// SIMATIC S7-200 SMART project (STEP 7-Micro/WIN SMART), CPU ST60

SYMBOL_TABLE V区符号
参数传输成功           V0.0     // 接收工控机传来的数据传输成功信号
参数是否更新           V0.1
挡板自动控制完成标志       V0.2
挡板电机开关           V0.3
挡板手动向内           V0.4
挡板手动向外           V0.5
置工件就绪            V0.6
下料电机开关           V0.7
下料前进点动           V1.0
下料后退点动           V1.1
冷却电机开关           V1.2
冷却电机向内           V1.3
冷却电机向外           V1.4
挡板电机查找原点按钮       V11.1
下料电机查找原点按钮       V11.2
冷却电机查找原点按钮       V11.3
挡板自动控制           V11.4
下料下移一个工位         V11.5
下料启动按钮           V11.6
下料手动完成标志         V11.7
回到底部             V12.0
冷却自动控制           V12.1
挡板电机初始化完成位       V20.1
挡板电机当前运动方向       V20.2
挡板电机查找原点完成位      V20.3
挡板电机GOTO完成位      V20.4
挡板电机错误参数         VB21
挡板电机当前位置         VD24
挡板电机当前速度         VD28
挡板电机移动位置         VD44
挡板电机速度           VD48
挡板电机移动模式         VB41
挡板电机停止运动轴        V40.1
挡板电机运动方向         V40.2
冷却电机初始化完成位       V60.1
冷却电机当前运动方向       V60.2
冷却电机查找原点完成位      V60.3
冷却电机GOTO完成位      V60.4
冷却电机错误参数         VB61
冷却电机当前位置         VD64
冷却电机当前速度         VD68
冷却电机移动位置         VD84
冷却电机速度           VD88
冷却电机移动模式         VB81
冷却电机停止运动轴        V80.1
冷却电机运动方向         V80.2
下料电机初始化完成位       V100.1
下料电机当前运动方向       V100.2
下料电机查找原点完成位      V100.3
下料电机GOTO完成位      V100.4
下料电机错误参数         VB101
下料电机当前位置         VD104
下料电机当前速度         VD108
下料电机移动位置         VD124
下料电机速度           VD128
下料电机移动模式         VB121
下料电机停止运动轴        V120.1
下料电机运动方向         V120.2
下料电机运动到杆件放置      VD150
下料电机下移一个杆件位      VD154
下料电机一号杆件位置       VD158
下料电机二号杆件位置       VD162
下料电机三号杆件位置       VD166
下料电机四号杆件位置       VD170
下料电机五号杆件位置       VD174
下料电机运动到下料位置      VD178
上一杆件数据           VD140
当前杆件数据           VD144
END_SYMBOL_TABLE

SYMBOL_TABLE 系统符号
Always_On        SM0.0    // 始终接通
END_SYMBOL_TABLE

SYMBOL_TABLE M区符号
挡板超限报警           M0.0     // 挡板的位置超过左右极限传感器的位置
更新配对表            M0.1
电机是否就绪状态位        M0.3
上料步进到位状态位        M0.4
上料工件有无状态位        M0.5
下料步进到位状态位        M0.6
下料小车到位状态位        M0.7
步进报警信息           M1.0
上料传动故障报警         M1.1
两次杆件之差           MD12
END_SYMBOL_TABLE

ORGANIZATION_BLOCK 主程序:OB1
TITLE=
BEGIN
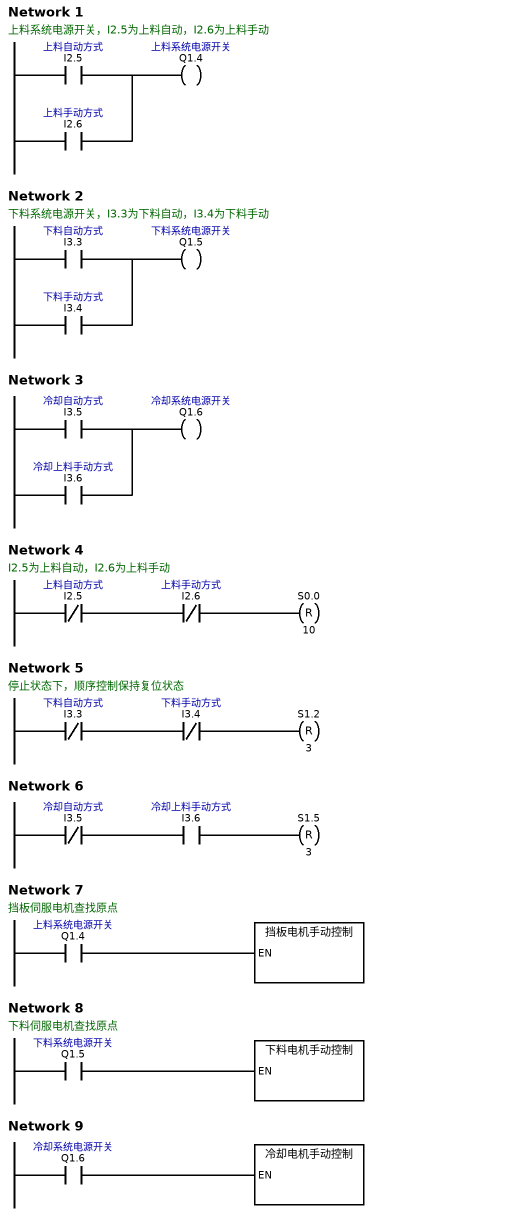
Network 1
// 上料系统电源开关，I2.5为上料自动，I2.6为上料手动
LD     上料自动方式:I2.5
O      上料手动方式:I2.6
=      上料系统电源开关:Q1.4
Network 2
// 下料系统电源开关，I3.3为下料自动，I3.4为下料手动
LD     下料自动方式:I3.3
O      下料手动方式:I3.4
=      下料系统电源开关:Q1.5
Network 3
LD     冷却自动方式:I3.5
O      冷却上料手动方式:I3.6
=      冷却系统电源开关:Q1.6
Network 4
// I2.5为上料自动，I2.6为上料手动
LDN    上料自动方式:I2.5
AN     上料手动方式:I2.6
R      S0.0, 10
Network 5
// 停止状态下，顺序控制保持复位状态
LDN    下料自动方式:I3.3
AN     下料手动方式:I3.4
R      S1.2, 3
Network 6
LDN    冷却自动方式:I3.5
A      冷却上料手动方式:I3.6
R      S1.5, 3
Network 7
// 挡板伺服电机查找原点
LD     上料系统电源开关:Q1.4
CALL   挡板电机手动控制:SBR7
Network 8
// 下料伺服电机查找原点
LD     下料系统电源开关:Q1.5
CALL   下料电机手动控制:SBR9
Network 9
LD     冷却系统电源开关:Q1.6
CALL   冷却电机手动控制:SBR18
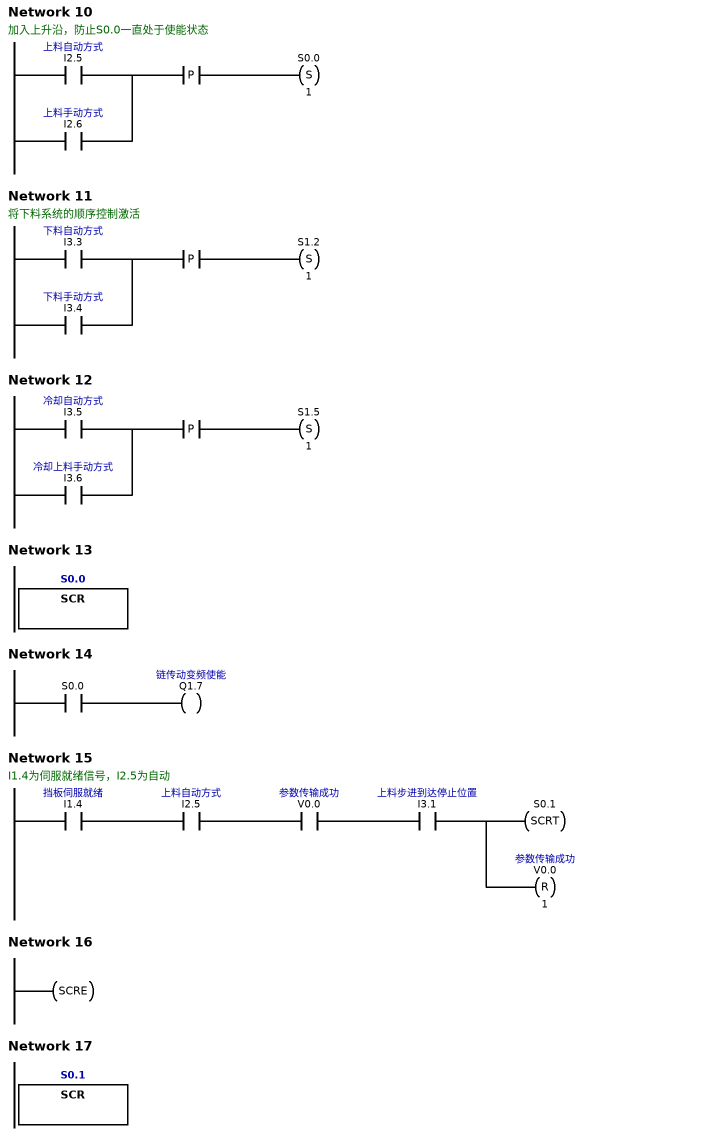
Network 10
// 加入上升沿，防止S0.0一直处于使能状态
LD     上料自动方式:I2.5
O      上料手动方式:I2.6
EU
S      S0.0, 1
Network 11
// 将下料系统的顺序控制激活
LD     下料自动方式:I3.3
O      下料手动方式:I3.4
EU
S      S1.2, 1
Network 12
LD     冷却自动方式:I3.5
O      冷却上料手动方式:I3.6
EU
S      S1.5, 1
Network 13
LSCR   S0.0
Network 14
LD     S0.0
=      链传动变频使能:Q1.7
Network 15
// I1.4为伺服就绪信号，I2.5为自动
LD     挡板伺服就绪:I1.4
A      上料自动方式:I2.5
A      参数传输成功:V0.0
A      上料步进到达停止位置:I3.1
SCRT   S0.1
R      参数传输成功:V0.0, 1
Network 16
SCRE
Network 17
LSCR   S0.1
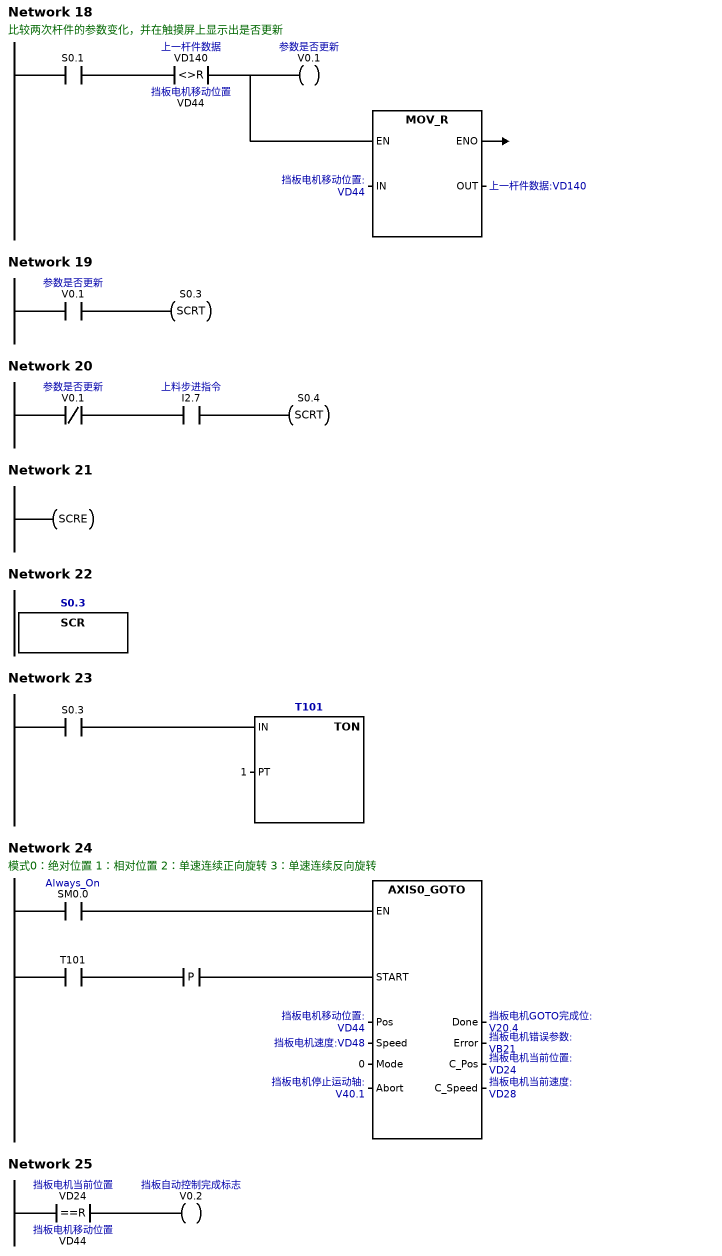
Network 18
// 比较两次杆件的参数变化，并在触摸屏上显示出是否更新
LD     S0.1
AR<>   上一杆件数据:VD140, 挡板电机移动位置:VD44
=      参数是否更新:V0.1
MOVR   挡板电机移动位置:VD44, 上一杆件数据:VD140
Network 19
LD     参数是否更新:V0.1
SCRT   S0.3
Network 20
LDN    参数是否更新:V0.1
A      上料步进指令:I2.7
SCRT   S0.4
Network 21
SCRE
Network 22
LSCR   S0.3
Network 23
LD     S0.3
TON    T101, 1
Network 24
// 模式0：绝对位置 1：相对位置 2：单速连续正向旋转 3：单速连续反向旋转
LD     Always_On:SM0.0
=      L60.0
LD     T101
EU
=      L63.7
LD     L60.0
CALL   AXIS0_GOTO:SBR4, L63.7, 挡板电机移动位置:VD44, 挡板电机速度:VD48, 0, 挡板电机停止运动轴:V40.1, 挡板电机GOTO完成位:V20.4, 挡板电机错误参数:VB21, 挡板电机当前位置:VD24, 挡板电机当前速度:VD28
Network 25
LDR=   挡板电机当前位置:VD24, 挡板电机移动位置:VD44
=      挡板自动控制完成标志:V0.2
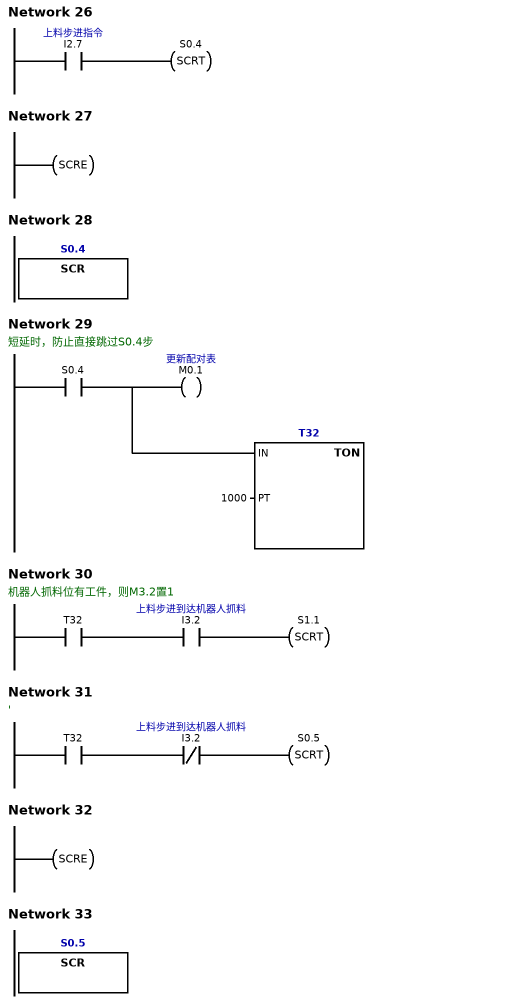
Network 26
LD     上料步进指令:I2.7
SCRT   S0.4
Network 27
SCRE
Network 28
LSCR   S0.4
Network 29
// 短延时，防止直接跳过S0.4步
LD     S0.4
=      更新配对表:M0.1
TON    T32, 1000
Network 30
// 机器人抓料位有工件，则M3.2置1
LD     T32
A      上料步进到达机器人抓料:I3.2
SCRT   S1.1
Network 31
// '
LD     T32
AN     上料步进到达机器人抓料:I3.2
SCRT   S0.5
Network 32
SCRE
Network 33
LSCR   S0.5
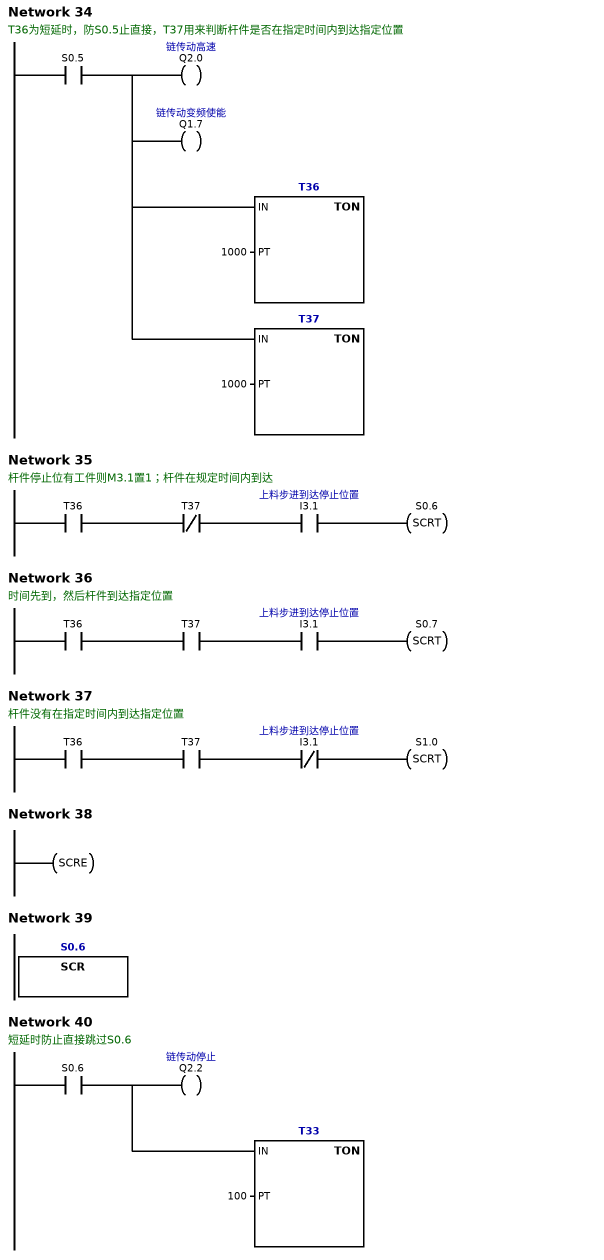
Network 34
// T36为短延时，防S0.5止直接，T37用来判断杆件是否在指定时间内到达指定位置
LD     S0.5
=      链传动高速:Q2.0
=      链传动变频使能:Q1.7
TON    T36, 1000
TON    T37, 1000
Network 35
// 杆件停止位有工件则M3.1置1；杆件在规定时间内到达
LD     T36
AN     T37
A      上料步进到达停止位置:I3.1
SCRT   S0.6
Network 36
// 时间先到，然后杆件到达指定位置
LD     T36
A      T37
A      上料步进到达停止位置:I3.1
SCRT   S0.7
Network 37
// 杆件没有在指定时间内到达指定位置
LD     T36
A      T37
AN     上料步进到达停止位置:I3.1
SCRT   S1.0
Network 38
SCRE
Network 39
LSCR   S0.6
Network 40
// 短延时防止直接跳过S0.6
LD     S0.6
=      链传动停止:Q2.2
TON    T33, 100
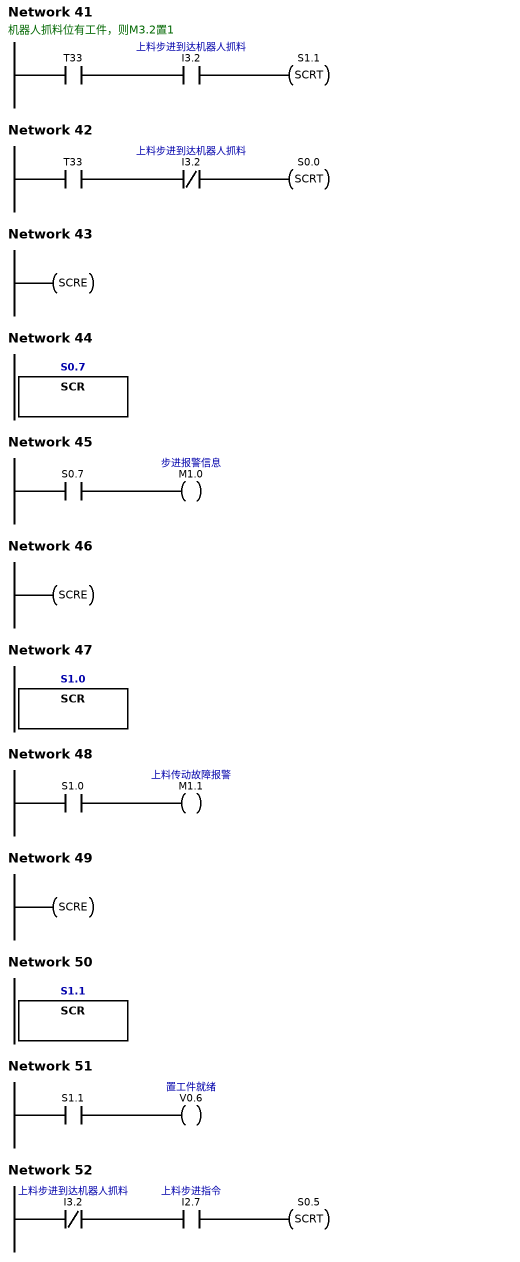
Network 41
// 机器人抓料位有工件，则M3.2置1
LD     T33
A      上料步进到达机器人抓料:I3.2
SCRT   S1.1
Network 42
LD     T33
AN     上料步进到达机器人抓料:I3.2
SCRT   S0.0
Network 43
SCRE
Network 44
LSCR   S0.7
Network 45
LD     S0.7
=      步进报警信息:M1.0
Network 46
SCRE
Network 47
LSCR   S1.0
Network 48
LD     S1.0
=      上料传动故障报警:M1.1
Network 49
SCRE
Network 50
LSCR   S1.1
Network 51
LD     S1.1
=      置工件就绪:V0.6
Network 52
LDN    上料步进到达机器人抓料:I3.2
A      上料步进指令:I2.7
SCRT   S0.5
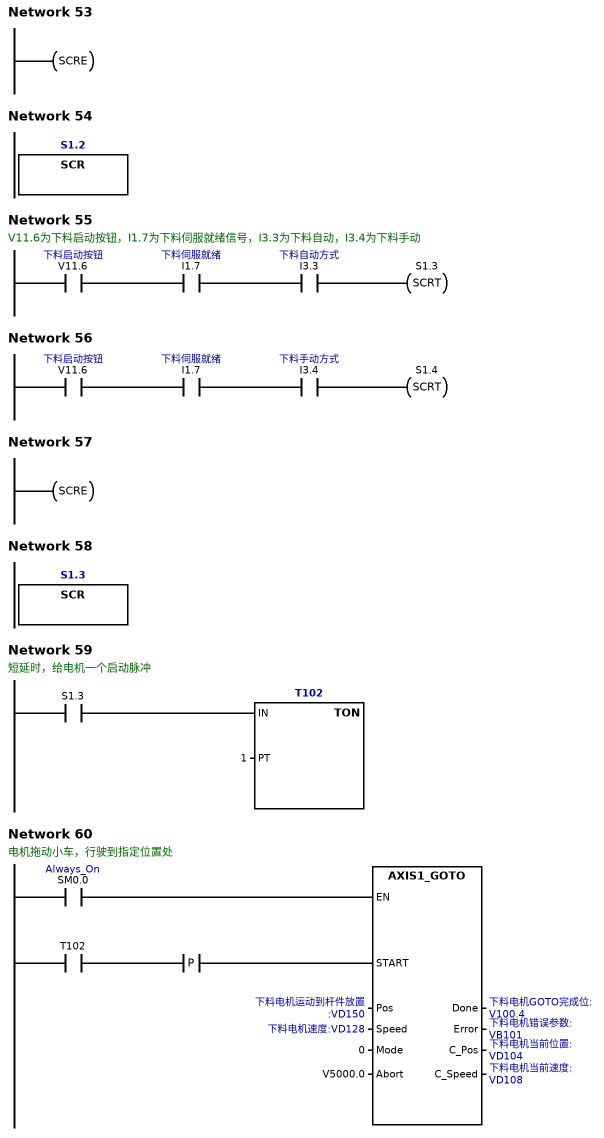
Network 53
SCRE
Network 54
LSCR   S1.2
Network 55
// V11.6为下料启动按钮，I1.7为下料伺服就绪信号，I3.3为下料自动，I3.4为下料手动
LD     下料启动按钮:V11.6
A      下料伺服就绪:I1.7
A      下料自动方式:I3.3
SCRT   S1.3
Network 56
LD     下料启动按钮:V11.6
A      下料伺服就绪:I1.7
A      下料手动方式:I3.4
SCRT   S1.4
Network 57
SCRE
Network 58
LSCR   S1.3
Network 59
// 短延时，给电机一个启动脉冲
LD     S1.3
TON    T102, 1
Network 60
// 电机拖动小车，行驶到指定位置处
LD     Always_On:SM0.0
=      L60.0
LD     T102
EU
=      L63.7
LD     L60.0
CALL   AXIS1_GOTO:SBR11, L63.7, 下料电机运动到杆件放置:VD150, 下料电机速度:VD128, 0, V5000.0, 下料电机GOTO完成位:V100.4, 下料电机错误参数:VB101, 下料电机当前位置:VD104, 下料电机当前速度:VD108
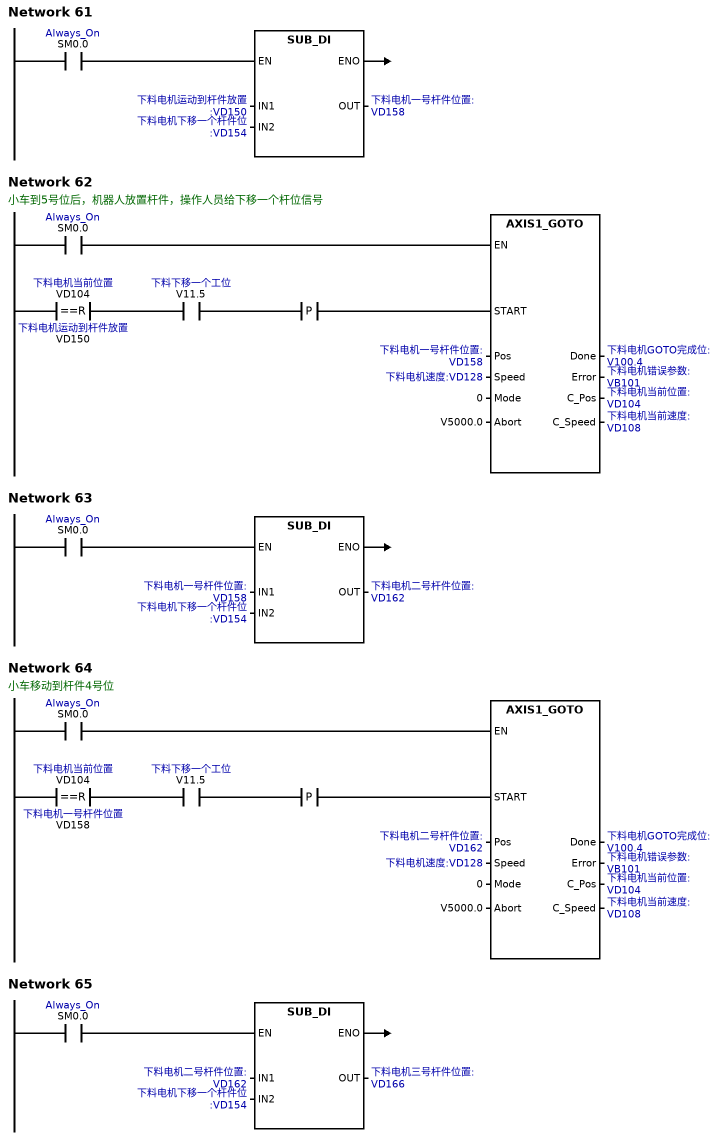
Network 61
LD     Always_On:SM0.0
MOVD   下料电机运动到杆件放置:VD150, 下料电机一号杆件位置:VD158
-D     下料电机下移一个杆件位:VD154, 下料电机一号杆件位置:VD158
Network 62
// 小车到5号位后，机器人放置杆件，操作人员给下移一个杆位信号
LD     Always_On:SM0.0
=      L60.0
LDR=   下料电机当前位置:VD104, 下料电机运动到杆件放置:VD150
A      下料下移一个工位:V11.5
EU
=      L63.7
LD     L60.0
CALL   AXIS1_GOTO:SBR11, L63.7, 下料电机一号杆件位置:VD158, 下料电机速度:VD128, 0, V5000.0, 下料电机GOTO完成位:V100.4, 下料电机错误参数:VB101, 下料电机当前位置:VD104, 下料电机当前速度:VD108
Network 63
LD     Always_On:SM0.0
MOVD   下料电机一号杆件位置:VD158, 下料电机二号杆件位置:VD162
-D     下料电机下移一个杆件位:VD154, 下料电机二号杆件位置:VD162
Network 64
// 小车移动到杆件4号位
LD     Always_On:SM0.0
=      L60.0
LDR=   下料电机当前位置:VD104, 下料电机一号杆件位置:VD158
A      下料下移一个工位:V11.5
EU
=      L63.7
LD     L60.0
CALL   AXIS1_GOTO:SBR11, L63.7, 下料电机二号杆件位置:VD162, 下料电机速度:VD128, 0, V5000.0, 下料电机GOTO完成位:V100.4, 下料电机错误参数:VB101, 下料电机当前位置:VD104, 下料电机当前速度:VD108
Network 65
LD     Always_On:SM0.0
MOVD   下料电机二号杆件位置:VD162, 下料电机三号杆件位置:VD166
-D     下料电机下移一个杆件位:VD154, 下料电机三号杆件位置:VD166
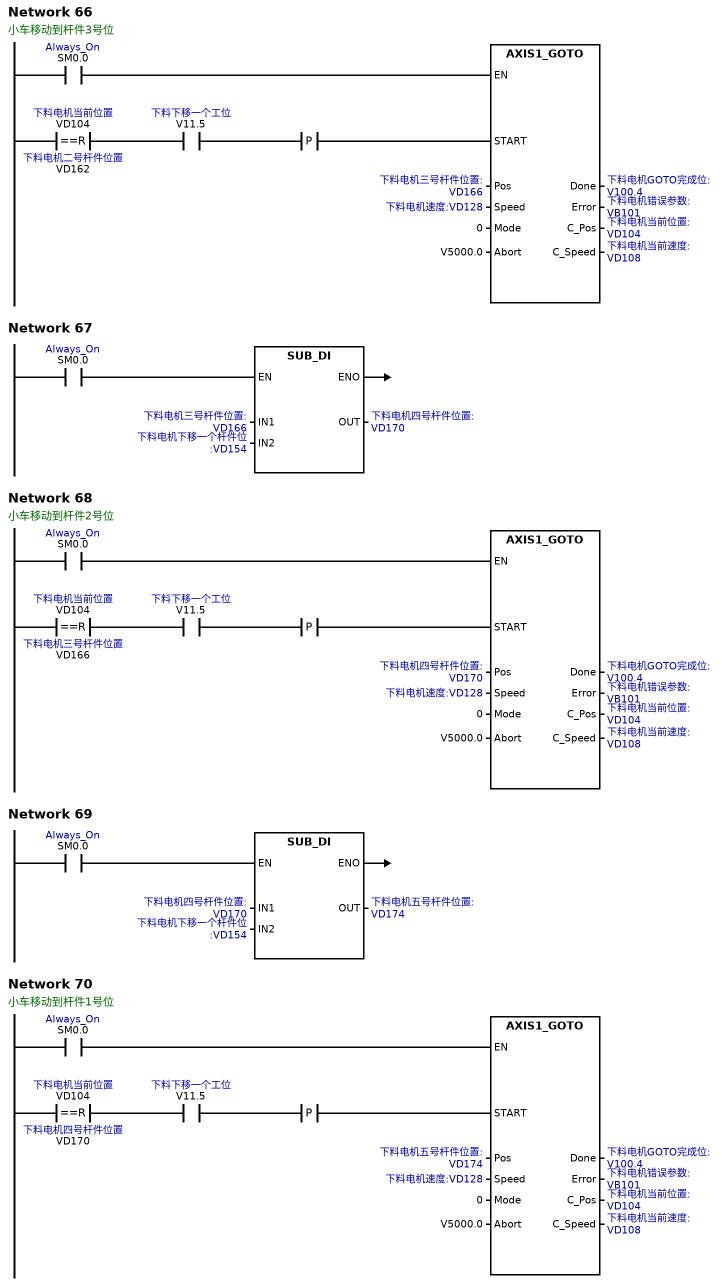
Network 66
// 小车移动到杆件3号位
LD     Always_On:SM0.0
=      L60.0
LDR=   下料电机当前位置:VD104, 下料电机二号杆件位置:VD162
A      下料下移一个工位:V11.5
EU
=      L63.7
LD     L60.0
CALL   AXIS1_GOTO:SBR11, L63.7, 下料电机三号杆件位置:VD166, 下料电机速度:VD128, 0, V5000.0, 下料电机GOTO完成位:V100.4, 下料电机错误参数:VB101, 下料电机当前位置:VD104, 下料电机当前速度:VD108
Network 67
LD     Always_On:SM0.0
MOVD   下料电机三号杆件位置:VD166, 下料电机四号杆件位置:VD170
-D     下料电机下移一个杆件位:VD154, 下料电机四号杆件位置:VD170
Network 68
// 小车移动到杆件2号位
LD     Always_On:SM0.0
=      L60.0
LDR=   下料电机当前位置:VD104, 下料电机三号杆件位置:VD166
A      下料下移一个工位:V11.5
EU
=      L63.7
LD     L60.0
CALL   AXIS1_GOTO:SBR11, L63.7, 下料电机四号杆件位置:VD170, 下料电机速度:VD128, 0, V5000.0, 下料电机GOTO完成位:V100.4, 下料电机错误参数:VB101, 下料电机当前位置:VD104, 下料电机当前速度:VD108
Network 69
LD     Always_On:SM0.0
MOVD   下料电机四号杆件位置:VD170, 下料电机五号杆件位置:VD174
-D     下料电机下移一个杆件位:VD154, 下料电机五号杆件位置:VD174
Network 70
// 小车移动到杆件1号位
LD     Always_On:SM0.0
=      L60.0
LDR=   下料电机当前位置:VD104, 下料电机四号杆件位置:VD170
A      下料下移一个工位:V11.5
EU
=      L63.7
LD     L60.0
CALL   AXIS1_GOTO:SBR11, L63.7, 下料电机五号杆件位置:VD174, 下料电机速度:VD128, 0, V5000.0, 下料电机GOTO完成位:V100.4, 下料电机错误参数:VB101, 下料电机当前位置:VD104, 下料电机当前速度:VD108
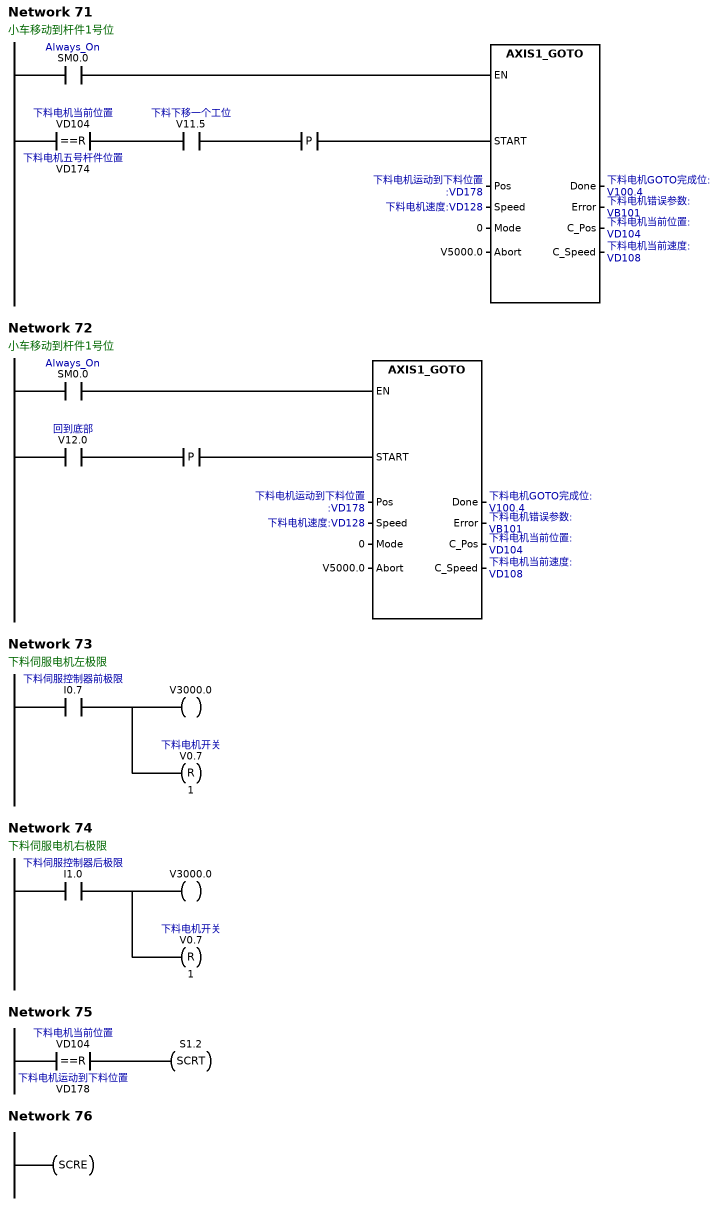
Network 71
// 小车移动到杆件1号位
LD     Always_On:SM0.0
=      L60.0
LDR=   下料电机当前位置:VD104, 下料电机五号杆件位置:VD174
A      下料下移一个工位:V11.5
EU
=      L63.7
LD     L60.0
CALL   AXIS1_GOTO:SBR11, L63.7, 下料电机运动到下料位置:VD178, 下料电机速度:VD128, 0, V5000.0, 下料电机GOTO完成位:V100.4, 下料电机错误参数:VB101, 下料电机当前位置:VD104, 下料电机当前速度:VD108
Network 72
// 小车移动到杆件1号位
LD     Always_On:SM0.0
=      L60.0
LD     回到底部:V12.0
EU
=      L63.7
LD     L60.0
CALL   AXIS1_GOTO:SBR11, L63.7, 下料电机运动到下料位置:VD178, 下料电机速度:VD128, 0, V5000.0, 下料电机GOTO完成位:V100.4, 下料电机错误参数:VB101, 下料电机当前位置:VD104, 下料电机当前速度:VD108
Network 73
// 下料伺服电机左极限
LD     下料伺服控制器前极限:I0.7
=      V3000.0
R      下料电机开关:V0.7, 1
Network 74
// 下料伺服电机右极限
LD     下料伺服控制器后极限:I1.0
=      V3000.0
R      下料电机开关:V0.7, 1
Network 75
LDR=   下料电机当前位置:VD104, 下料电机运动到下料位置:VD178
SCRT   S1.2
Network 76
SCRE
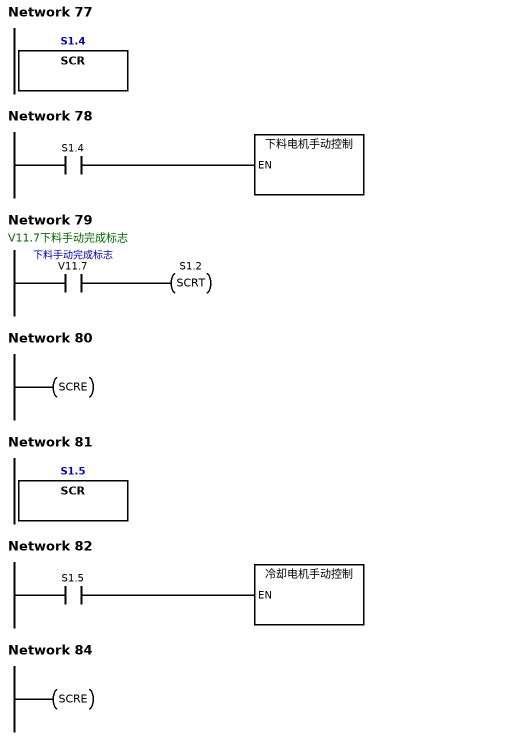
Network 77
LSCR   S1.4
Network 78
LD     S1.4
CALL   下料电机手动控制:SBR9
Network 79
// V11.7下料手动完成标志
LD     下料手动完成标志:V11.7
SCRT   S1.2
Network 80
SCRE
Network 81
LSCR   S1.5
Network 82
LD     S1.5
CALL   冷却电机手动控制:SBR18
Network 84
SCRE
END_ORGANIZATION_BLOCK

// SBR2: protected block, not included

// SBR3: protected block, not included

// SBR4: protected block, not included

// SBR5: protected block, not included

// SBR6: protected block, not included

SUBROUTINE_BLOCK 挡板电机手动控制:SBR7
TITLE=子程序注释
BEGIN
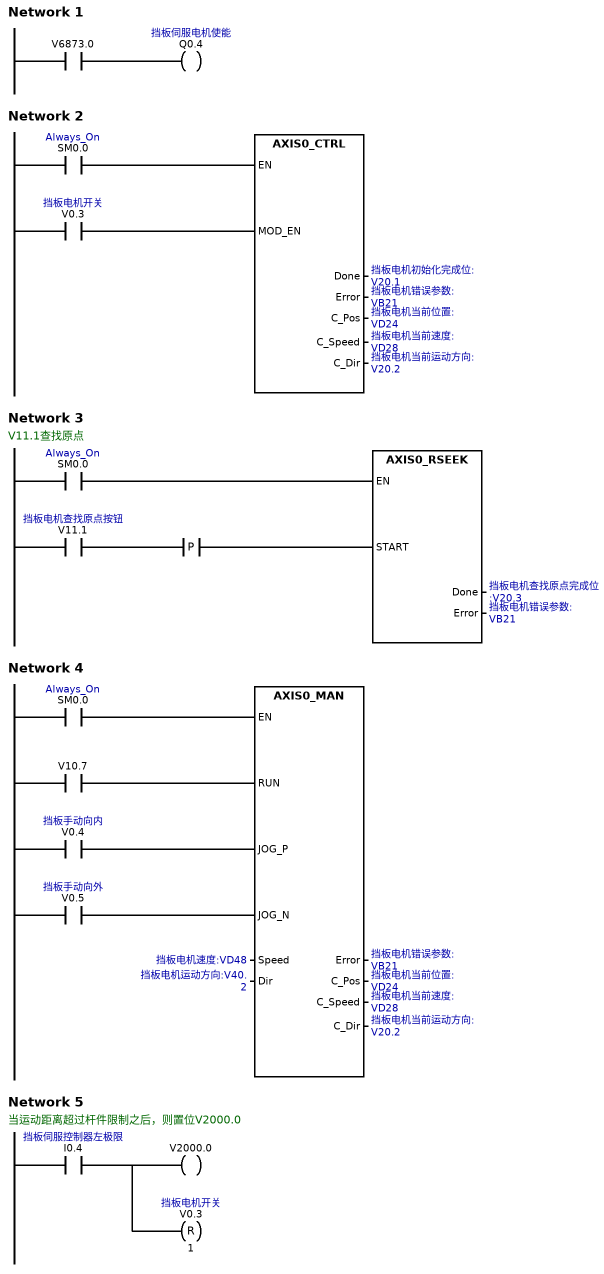
Network 1
LD     V6873.0
=      挡板伺服电机使能:Q0.4
Network 2
LD     Always_On:SM0.0
=      L60.0
LD     挡板电机开关:V0.3
=      L63.7
LD     L60.0
CALL   AXIS0_CTRL:SBR2, L63.7, 挡板电机初始化完成位:V20.1, 挡板电机错误参数:VB21, 挡板电机当前位置:VD24, 挡板电机当前速度:VD28, 挡板电机当前运动方向:V20.2
Network 3
// V11.1查找原点
LD     Always_On:SM0.0
=      L60.0
LD     挡板电机查找原点按钮:V11.1
EU
=      L63.7
LD     L60.0
CALL   AXIS0_RSEEK:SBR5, L63.7, 挡板电机查找原点完成位:V20.3, 挡板电机错误参数:VB21
Network 4
LD     Always_On:SM0.0
=      L60.0
LD     V10.7
=      L63.7
LD     挡板手动向内:V0.4
=      L63.6
LD     挡板手动向外:V0.5
=      L63.5
LD     L60.0
CALL   AXIS0_MAN:SBR3, L63.7, L63.6, L63.5, 挡板电机速度:VD48, 挡板电机运动方向:V40.2, 挡板电机错误参数:VB21, 挡板电机当前位置:VD24, 挡板电机当前速度:VD28, 挡板电机当前运动方向:V20.2
Network 5
// 当运动距离超过杆件限制之后，则置位V2000.0
LD     挡板伺服控制器左极限:I0.4
=      V2000.0
R      挡板电机开关:V0.3, 1
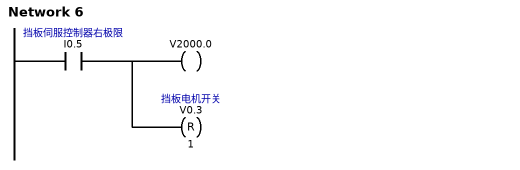
Network 6
LD     挡板伺服控制器右极限:I0.5
=      V2000.0
R      挡板电机开关:V0.3, 1
END_SUBROUTINE_BLOCK

SUBROUTINE_BLOCK 下料电机手动控制:SBR9
TITLE=子程序注释
BEGIN
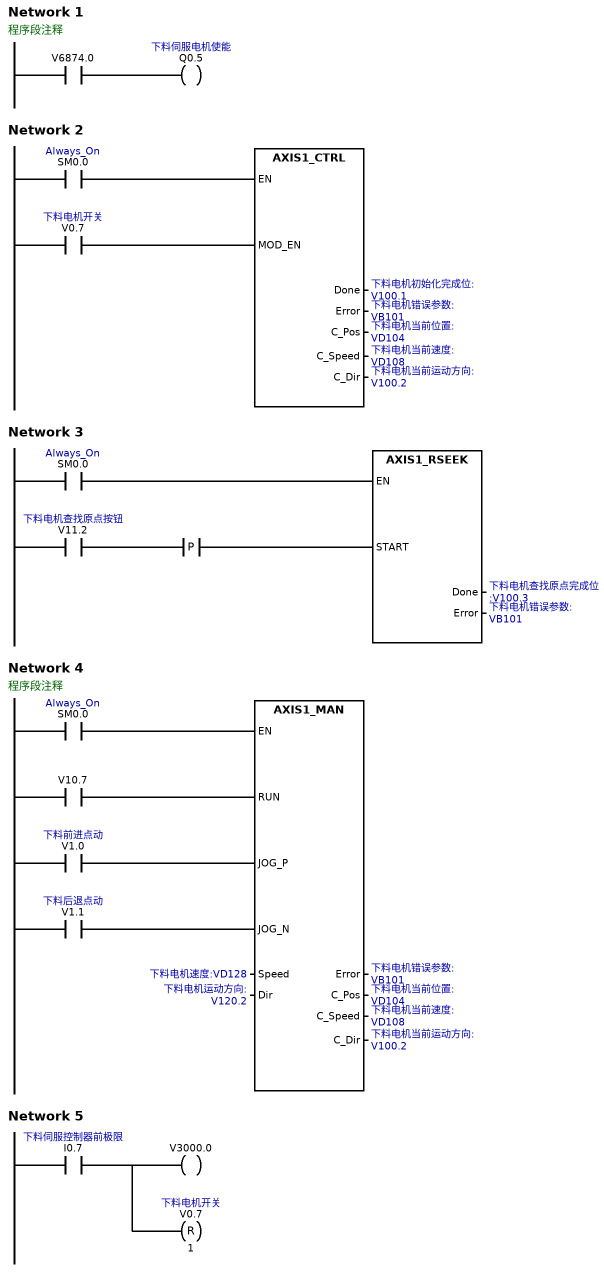
Network 1
// 程序段注释
LD     V6874.0
=      下料伺服电机使能:Q0.5
Network 2
LD     Always_On:SM0.0
=      L60.0
LD     下料电机开关:V0.7
=      L63.7
LD     L60.0
CALL   AXIS1_CTRL:SBR6, L63.7, 下料电机初始化完成位:V100.1, 下料电机错误参数:VB101, 下料电机当前位置:VD104, 下料电机当前速度:VD108, 下料电机当前运动方向:V100.2
Network 3
LD     Always_On:SM0.0
=      L60.0
LD     下料电机查找原点按钮:V11.2
EU
=      L63.7
LD     L60.0
CALL   AXIS1_RSEEK:SBR12, L63.7, 下料电机查找原点完成位:V100.3, 下料电机错误参数:VB101
Network 4
// 程序段注释
LD     Always_On:SM0.0
=      L60.0
LD     V10.7
=      L63.7
LD     下料前进点动:V1.0
=      L63.6
LD     下料后退点动:V1.1
=      L63.5
LD     L60.0
CALL   AXIS1_MAN:SBR10, L63.7, L63.6, L63.5, 下料电机速度:VD128, 下料电机运动方向:V120.2, 下料电机错误参数:VB101, 下料电机当前位置:VD104, 下料电机当前速度:VD108, 下料电机当前运动方向:V100.2
Network 5
LD     下料伺服控制器前极限:I0.7
=      V3000.0
R      下料电机开关:V0.7, 1
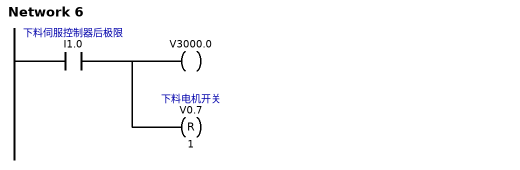
Network 6
LD     下料伺服控制器后极限:I1.0
=      V3000.0
R      下料电机开关:V0.7, 1
END_SUBROUTINE_BLOCK

// SBR10: protected block, not included

// SBR11: protected block, not included

// SBR12: protected block, not included

// SBR13: protected block, not included

// SBR14: protected block, not included

// SBR15: protected block, not included

// SBR16: protected block, not included

SUBROUTINE_BLOCK 冷却电机手动控制:SBR18
TITLE=子程序注释
BEGIN
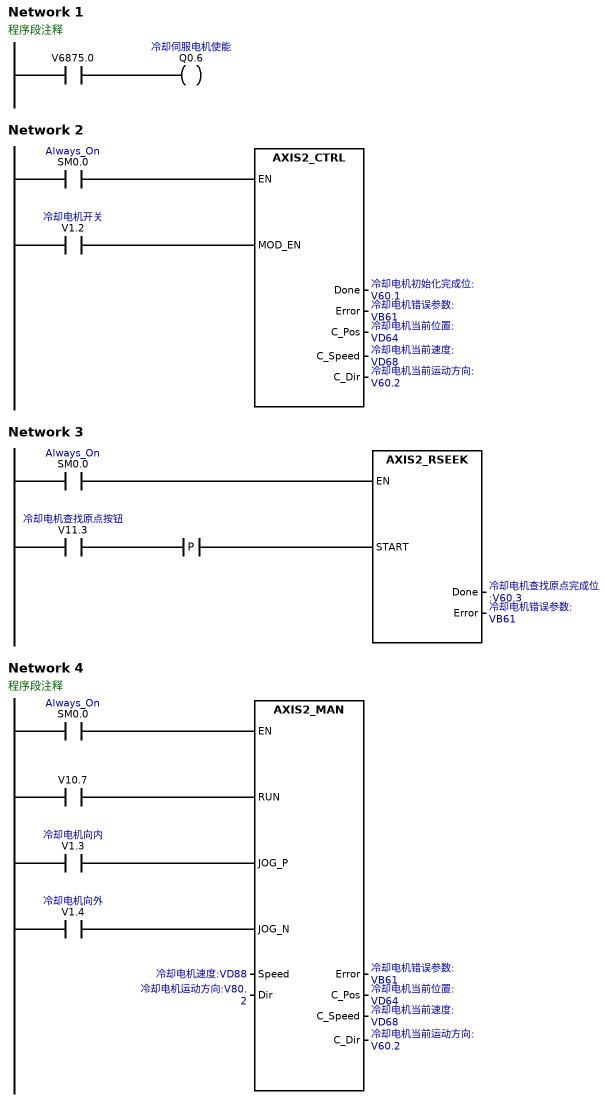
Network 1
// 程序段注释
LD     V6875.0
=      冷却伺服电机使能:Q0.6
Network 2
LD     Always_On:SM0.0
=      L60.0
LD     冷却电机开关:V1.2
=      L63.7
LD     L60.0
CALL   AXIS2_CTRL:SBR13, L63.7, 冷却电机初始化完成位:V60.1, 冷却电机错误参数:VB61, 冷却电机当前位置:VD64, 冷却电机当前速度:VD68, 冷却电机当前运动方向:V60.2
Network 3
LD     Always_On:SM0.0
=      L60.0
LD     冷却电机查找原点按钮:V11.3
EU
=      L63.7
LD     L60.0
CALL   AXIS2_RSEEK:SBR16, L63.7, 冷却电机查找原点完成位:V60.3, 冷却电机错误参数:VB61
Network 4
// 程序段注释
LD     Always_On:SM0.0
=      L60.0
LD     V10.7
=      L63.7
LD     冷却电机向内:V1.3
=      L63.6
LD     冷却电机向外:V1.4
=      L63.5
LD     L60.0
CALL   AXIS2_MAN:SBR14, L63.7, L63.6, L63.5, 冷却电机速度:VD88, 冷却电机运动方向:V80.2, 冷却电机错误参数:VB61, 冷却电机当前位置:VD64, 冷却电机当前速度:VD68, 冷却电机当前运动方向:V60.2
END_SUBROUTINE_BLOCK
